ABB RAPID module: Assignment2.mod

MODULE Assignment2

    VAR socketdev client_socket;
    ! The host and port that we will be listening for a connection on.
    !PERS string host := "127.0.0.1";

    VAR num effectorHeight:= 147;
    VAR robtarget testTarget := [[175, -100, 147],[0,0,-1,0],[0,0,0,0],[9E+09,9E+09,9E+09,9E+09,9E+09,9E+09]];

    VAR num jog_inc:=30;
    VAR num jog_inc_deg:= 5;
    VAR speeddata jog_speed:=v100;
    VAR speeddata pose_speed:= v100;
    PERS string current_state := "None";
    PERS bool quit := FALSE;
    PERS bool done := FALSE;
    PERS bool checkCom := FALSE;
    !VAR num numEnd;
    !VAR num numStart;
    !VAR string numTotal;


    ! The Main procedure. When you select 'PP to Main' on the FlexPendant, it will go to this procedure.
    PROC Main()

        !this is just for testing
        !numEnd := strLen("jogX 60");
        !numStart :=strFind("jogX 60",1,STR_DIGIT);
        !numTotal := strPart("jogX 60",numStart,numEnd-numStart+1);
        MoveToCalibPos;
    WHILE quit = FALSE DO
        WaitUntil checkCom = TRUE;
        !only use this if the position can deviate to avoid singularities
        SingArea \Wrist;

        !absolute position
        confj  \On;

        VelSet 70, 800;
        IF current_state <> "cancel" THEN
            IF current_state = "xPlus" THEN
                JogX(jog_inc);
                done:= TRUE;
                current_state := "None";
                WaitTime 2;
            ENDIF
            IF current_state = "yPlus" THEN
                JogY(jog_inc);
                done:=TRUE;
                current_state := "None";
                WaitTime 2;
            ENDIF
            IF current_state = "zPlus" THEN
                JogZ(jog_inc);
                done:=TRUE;
                current_state := "None";
                WaitTime 2;
            ENDIF
            IF current_state = "xMinus" THEN
                JogX(-jog_inc);
                done:=TRUE;
                current_state := "None";
                WaitTime 2;
            ENDIF
            IF current_state = "yMinus" THEN
                JogY(-jog_inc);
                done:=TRUE;
                current_state := "None";
                WaitTime 2;
            ENDIF
            IF current_state = "zMinus" THEN
                JogZ(-jog_inc);
                done:=TRUE;
                current_state := "None";
                WaitTime 2;
            ENDIF
            IF current_state = "jog1" THEN
                Jog1(jog_inc_deg);
                done:=TRUE;
                current_state := "None";
                WaitTime 2;
            ENDIF
            IF current_state = "conOn" THEN
                conRunOn;
                done:=TRUE;
                current_state := "None";
                WaitTime 2;
            ENDIF
            IF current_state = "conOff" THEN
                conRunOff;
                done:=TRUE;
                current_state := "None";
                WaitTime 2;
            ENDIF
            IF current_state = "conReverseOn" THEN
                conDirHome;
                done:=TRUE;
                current_state := "None";
                WaitTime 2;
            ENDIF
            IF current_state = "conReverseOff" THEN
                conDirRob;
                done:=TRUE;
                current_state := "None";
                WaitTime 2;
            ENDIF
            IF current_state = "vacSolOn" THEN
                vacSolOn;
                done:=TRUE;
                current_state := "None";
                WaitTime 2;
            ENDIF
            IF current_state = "vacSolOff" THEN
                vacSolOff;
                done:=TRUE;
                current_state := "None";
                WaitTime 2;
            ENDIF
            IF current_state = "vacPumpOn" THEN
                vacPwrOn;
                done:=TRUE;
                current_state := "None";
                WaitTime 2;
            ENDIF
            IF current_state = "vacPumpOff" THEN
                vacPwrOff;
                done:=TRUE;
                current_state := "None";
                WaitTime 2;
            ENDIF
            IF current_state = "paused" THEN
                StopMove;
                done:=TRUE;
                current_state := "None";
                WaitTime 2;
            ENDIF
            IF current_state = "resume" THEN
                StartMove;
                done:=TRUE;
                current_state := "None";
                WaitTime 2;
            ENDIF
            IF current_state = "quit" THEN
                quit:=TRUE;
                done:=TRUE;
                current_state := "None";
                WaitTime 2;
            ENDIF
            !ELSEIF current_state = "moveToPose" THEN
                !moveToPose(thetas_new);
                !WaitTime 2;
            !ELSEIF current_state = "moveAngle" THEN
                !moveAngle(robot_ang,robot_speed);
                !WaitTIme 2;
            IF current_state = "unknown" THEN
                TPWrite "Unknown command";
                WaitTime 2;
            ENDIF
        ELSE
        done:= TRUE;
        current_state := "None";
        WaitTime 2;
        ENDIF
        checkCom := FALSE;
    ENDWHILE

    ENDPROC

    PROC JogX(num jog_inc)
        VAR robtarget pos_current;
        VAR robtarget pos_new;
        VAR jointtarget jog_target;
        VAR errnum err_val;
        !get current pos
        pos_current:=CRobT();

        !calculate new pos
        pos_new:=pos_current;
        pos_new.trans.x:=pos_current.trans.x+jog_inc;

        jog_target:=CalcJointT(pos_new,tSCup,\ErrorNumber:=err_val);
        IF err_val=1135 OR err_val=1074 THEN
            !send message to matlab
            WaitTime 1;
        ELSE
            !move to calculated pos
            MoveL pos_new,jog_speed,fine,tSCup;
        ENDIF
    ENDPROC

    PROC JogY(num jog_inc)
        VAR robtarget pos_current;
        VAR robtarget pos_new;
        VAR jointtarget jog_target;
        VAR errnum err_val;
        !get current pos
        pos_current:=CRobT();
        !calculate new pos
        pos_new:=pos_current;
        pos_new.trans.y:=pos_current.trans.y+jog_inc;
        !check if reachable
        jog_target:=CalcJointT(pos_new,tSCup,\ErrorNumber:=err_val);
        IF err_val=1135 OR err_val=1074 THEN
            !send message to matlab
            WaitTime 1;
        ELSE
            !move to calculated pos
            MoveL pos_new,jog_speed,fine,tSCup;
        ENDIF
    ENDPROC

    PROC JogZ(num jog_inc)
        VAR robtarget pos_current;
        VAR robtarget pos_new;
        VAR jointtarget jog_target;
        VAR errnum err_val;
        !get current pos
        pos_current:=CRobT();

        !calculate new pos
        pos_new:=pos_current;
        pos_new.trans.z:=pos_current.trans.z+jog_inc;

        jog_target:=CalcJointT(pos_new,tSCup,\ErrorNumber:=err_val);
        IF err_val=1135 OR err_val=1074 THEN
            !send message to matlab
            WaitTime 1;
        ELSE
            !move to calculated pos
            MoveL pos_new,jog_speed,fine,tSCup;
        ENDIF
    ENDPROC

    !Jog Joint 1
    PROC Jog1(num jog_inc_deg)
        VAR jointtarget thetas_current;
        VAR jointtarget thetas_new;
        VAR robtarget pos_new;
        VAR errnum err_val;

        !get current
        thetas_current:=CJointT();
        thetas_new:=thetas_current;
        !increment new
        thetas_new.robax.rax_1:=thetas_new.robax.rax_1+jog_inc_deg;

        pos_new:=CalcRobT(thetas_new,tSCup);
        thetas_current:=CalcJointT(pos_new,tSCup,\ErrorNumber:=err_val);
        IF err_val=1135 OR err_val=1074 OR err_val = ERR_ROBLIMIT THEN
            !send message to matlab, out of range
        ELSE
            MoveAbsJ thetas_new,jog_speed,fine,tSCup;
            !send mesage to matlab
        ENDIF
    ENDPROC



     PROC MoveToPose(robjoint thetas_new)
        VAR jointtarget thetas_new_formatted;
        thetas_new_formatted:= [thetas_new, [9E+09,9E+09,9E+09,9E+09,9E+09,9E+09]];!the formatted joint angles for moving the robot


        MoveAbsJ thetas_new_formatted, jog_speed, fine, tSCup;

    ENDPROC


    PROC MoveAngle(robjoint robot_ang,speeddata robot_speed)
        VAR jointtarget lin_joint;
        VAR jointtarget jointpos;
        VAR robtarget ang_rob;
        VAR errnum myerrnum;
        jointpos:=[robot_ang,[9E+09,9E+09,9E+09,9E+09,9E+09,9E+09]];
        ang_rob:=CalcRobT(jointpos,tSCup);
        lin_joint:=CalcJointT(ang_rob,tSCup\ErrorNumber:=myerrnum);
    ERROR
    ENDPROC


    PROC MoveTarget(robtarget target)

            ! 'MoveJ' executes a joint motion towards a robtarget. This is used to move the robot quickly from one point to another when that
            !   movement does not need to be in a straight line.
            ! 'pTableHome' is a robtarget defined in system module. The exact location of this on the table has been provided to you.
            ! 'v100' is a speeddata variable, and defines how fast the robot should move. The numbers is the speed in mm/sec, in this case 100mm/sec.
            ! 'fine' is a zonedata variable, and defines how close the robot should move to a point before executing its next command.
            !   'fine' means very close, other values such as 'z10' or 'z50', will move within 10mm and 50mm respectively before executing the next command.
            ! 'tSCup' is a tooldata variable. This has been defined in a system module, and represents the tip of the suction cup, telling the robot that we
            !   want to move this point to the specified robtarget. Please be careful about what tool you use, as using the incorrect tool will result in
            !   the robot not moving where you would expect it to. Generally you should be using
            MoveJ target, v100, fine, tSCup;

    ENDPROC

    PROC MoveTargetOffset(robtarget target, num x, num y, num z)

              MoveL Offs(target, x, y, z), v100, fine, tSCup;
    ENDPROC

    PROC vacPwrOn()
        SetDO DO10_1, 1;
    ENDPROC

    PROC vacPwrOff()
        SetDO DO10_1, 0;
    ENDPROC

    PROC vacSolOn()
        SetDO DO10_2, 1;
    ENDPROC

    PROC vacSolOff()
        SetDO DO10_2, 0;
    ENDPROC

    PROC conRunOn()
        SetDO DO10_3, 1;
    ENDPROC

    PROC conRunOff()
        SetDO DO10_3, 0;
    ENDPROC

    PROC conDirRob()
        SetDO DO10_4, 1;
    ENDPROC

    PROC conDirHome()
        SetDO DO10_4, 0;
    ENDPROC


ENDMODULE
